{attribute addProperty BoxType "EL1259-0000-0018"}
{attribute addProperty Id "StatusAT %I*Status_32B8CA62324"}
{attribute addProperty CRC "2110270805"}
{attribute addProperty SizeInBites "32"}
{attribute addProperty SizeInBytes "4"}
TYPE MTO_Inputs_Channel_7DC82D55 :
STRUCT
	{attribute addProperty Name "Status"}
	Status AT %I* : Status_32B8CA62;
END_STRUCT
END_TYPE

(* stored: Version 1.2.0.0, ProductVersion 3.1.4024.9
   DUT MTO_Inputs_Channel_7DC82D55: Id {5c5d1e23-7827-4ee5-981c-51f405c9af2c} *)
